(* CoDeSys 2.3 export: UDP_COMMUNICATION.EXP *)
(* Libraries: 05_Utilities\MPLCCommunication_Ethernet.lib 30.1.17 00:00:00, 11_System\SysLibSockets.lib 27.1.17 13:50:06, Internal\MPLCIntern_Communication_Ethernet.lib 30.1.17 00:00:00, standard.lib 27.1.17 13:50:06 *)

(* Global variable list: CodeSamples/UDP_Communication/UDP_Konstanten *)
VAR_GLOBAL CONSTANT
	UDP_CommAnzPD: INT := 64;  (*Datengröße in Byte*)
END_VAR
VAR_GLOBAL
END_VAR

(* POU CodeSamples/UDP_Communication/UDP_Communication_PRG, FBD *)
PROGRAM UDP_Communication_PRG
VAR
	bTest1: BOOL;
	bTest2: BOOL;
	bTest3: BOOL;
	fbUDP_Communication_MasterSlave: UDP_Communication_MasterSlave;
	bMaster: BOOL;
	nPort: UINT;
	sIP: STRING;
	tCycleTime: TIME;
	DataOUT: ARRAY[1..UDP_CommAnzPD] OF WORD;
	ttimeOut: TIME;
	DataIN: ARRAY[1..UDP_CommAnzPD] OF WORD;
END_VAR

(*Example inputs for MASTER---------------------------------------------------------------
UDP_Communication_MasterSlave(
	Enable:=TRUE , 
	SendMaster:=TRUE , 
	Port:= 44818, 
	IPAdr:= '10.1.254.129', 
	CycleTime:=t#100ms, 
	PE_Data:=fbUDP_Communication_MasterSlave.PE_Data , 
	TimeOut:=t#1000ms , 
	ChangeByteOrder:=FALSE , 
	Done=> , 
	Error=> , 
	ErrorID=> , 
	PDTimeOut=> , 
	PA_Data=> );

Example inputs for SLAVE---------------------------------------------------------------
UDP_Communication_MasterSlave(
	Enable:=TRUE , 
	SendMaster:=FALSE , 
	Port:= 44818, 
	IPAdr:= '10.1.254.128', 
	CycleTime:=t#100ms, 
	PE_Data:=fbUDP_Communication_MasterSlave.PE_Data , 
	TimeOut:=t#1000ms , 
	ChangeByteOrder:=FALSE , 
	Done=> , 
	Error=> , 
	ErrorID=> , 
	PDTimeOut=> , 
	PA_Data=> );
*)	
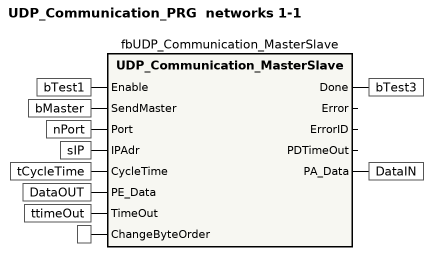
_FBD_ (* Function Block Diagram *)
NETWORK 1
	fbUDP_Communication_MasterSlave:UDP_Communication_MasterSlave(Enable: bTest1, SendMaster: bMaster, Port: nPort, IPAdr: sIP, CycleTime: tCycleTime, PE_Data: DataOUT, TimeOut: ttimeOut, ChangeByteOrder: , PA_Data => DataIN) => bTest3
_END_FBD_
END_PROGRAM

(* POU CodeSamples/UDP_Communication/UDP_Communication_MasterSlave, FBD *)
FUNCTION_BLOCK UDP_Communication_MasterSlave
VAR_INPUT
	Enable:BOOL;
	SendMaster : BOOL;  (* TRUE : Senden alle CycleTime, FALSE: Senden wenn ein Telegramm empfangen wurde *)
	Port:UINT;
	IPAdr:STRING(15);
	CycleTime :TIME;
	PE_Data:ARRAY[1..UDP_CommAnzPD] OF WORD;
	TimeOut:TIME;
	ChangeByteOrder : BOOL;
END_VAR
VAR_OUTPUT
	Done:BOOL;
	Error:BOOL;
	ErrorID:DWORD;
	PDTimeOut:BOOL;
	PA_Data:ARRAY[1..UDP_CommAnzPD] OF WORD;
END_VAR
VAR
	fbMC_ConnectV2_UDP: MC_ConnectV2_UDP;
	fbMC_ReceiveV2_UDP: MC_ReceiveV2_UDP;
	fbMC_SendV2_UDP: MC_SendV2_UDP;
	fbConvert_Array_1: WORDARRAY_TO_BYTEARRAY;
	fbConvert_Array: BYTEARRAY_TO_WORDARRAY_V2;
	R_TRIG_SendTrigger: R_TRIG;
	TON_TimeOut: TON;
	TON_CyclicSend: TON;

	refUDPConnection: MC_ConnectionV2_UDP;

	Send_Data_Array: ARRAY[0..1447] OF BYTE;
	Receive_Data_ArraY: ARRAY[0..1447] OF BYTE;


	bInitError: BOOL;
	nInitErrorID: DWORD;
	bSendError: BOOL;
	nSendErrorID: DWORD;
	bRecError: BOOL;
	nRecErrorID: DWORD;


	bCyclicSendTrigger: BOOL;
	bRecvDone: BOOL;

	nRxCounterOld: UINT;

END_VAR
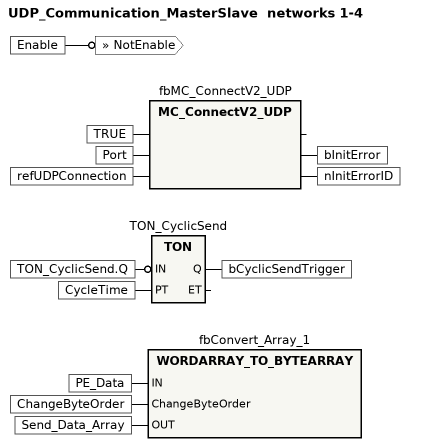
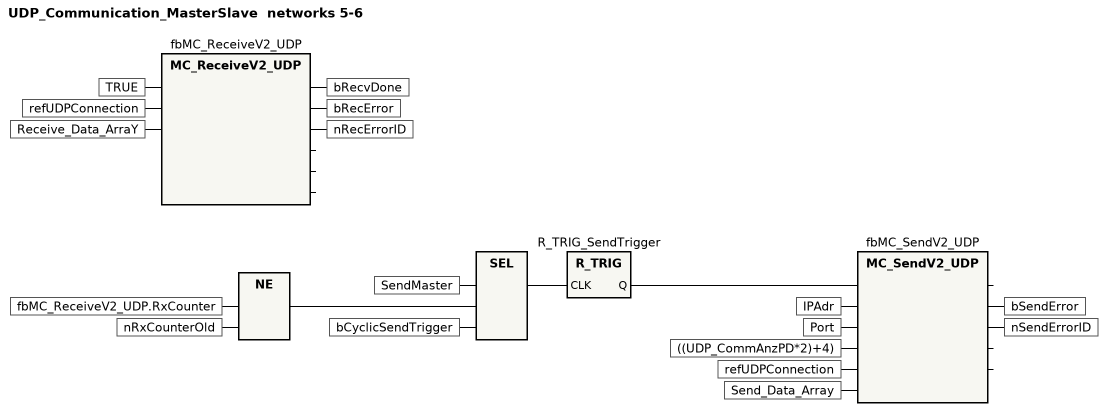
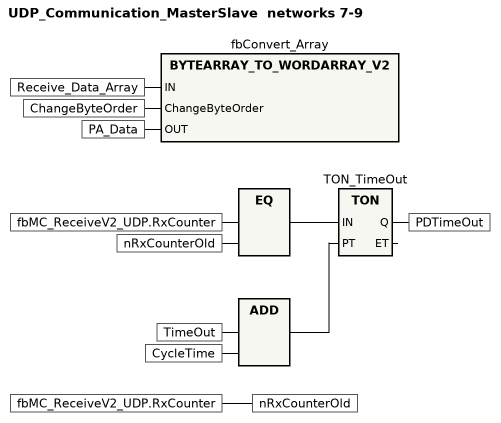
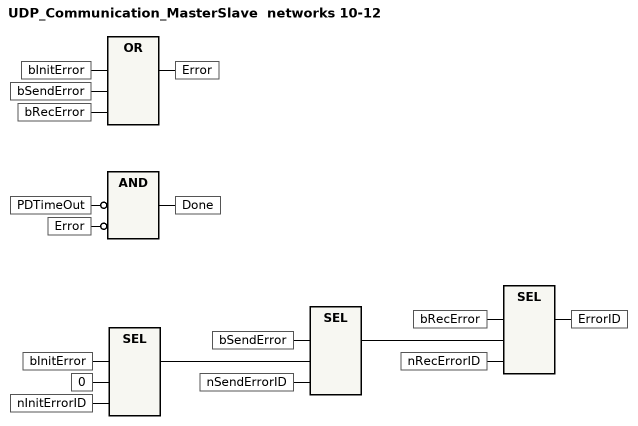
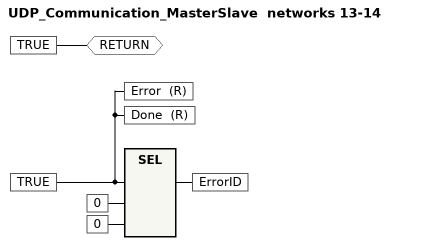
_FBD_ (* Function Block Diagram *)
NETWORK 1
	NOT Enable => >>NotEnable
NETWORK 2 (* Initialisierung der UDP-Kommunikation *)
	fbMC_ConnectV2_UDP:MC_ConnectV2_UDP(TRUE, Port, refUDPConnection, out 2 => bInitError, out 3 => nInitErrorID)
NETWORK 3 (* SendeTrigger für Senden wenn Master *)
	TON_CyclicSend:TON(IN: NOT TON_CyclicSend.Q, PT: CycleTime) => bCyclicSendTrigger
NETWORK 4 (* Umkopieren WORD-Array in BYTE-Array *)
	fbConvert_Array_1:WORDARRAY_TO_BYTEARRAY(IN: PE_Data, ChangeByteOrder: ChangeByteOrder, OUT: Send_Data_Array)
NETWORK 5 (* Daten empfangen über UDP *)
	fbMC_ReceiveV2_UDP:MC_ReceiveV2_UDP(TRUE, refUDPConnection, Receive_Data_ArraY, out 2 => bRecError, out 3 => nRecErrorID) => bRecvDone
NETWORK 6 (* Daten senden über UDP *)
	fbMC_SendV2_UDP:MC_SendV2_UDP(R_TRIG_SendTrigger:R_TRIG(CLK: SEL(SendMaster, NE(fbMC_ReceiveV2_UDP.RxCounter, nRxCounterOld), bCyclicSendTrigger)), IPAdr, Port, ((UDP_CommAnzPD*2)+4), refUDPConnection, Send_Data_Array, out 2 => bSendError, out 3 => nSendErrorID)
NETWORK 7 (* Konvertiere BYTE-Array in WORD-Array *)
	fbConvert_Array:BYTEARRAY_TO_WORDARRAY_V2(IN: Receive_Data_Array, ChangeByteOrder: ChangeByteOrder, OUT: PA_Data)
NETWORK 8
	TON_TimeOut:TON(IN: EQ(fbMC_ReceiveV2_UDP.RxCounter, nRxCounterOld), PT: ADD(TimeOut, CycleTime)) => PDTimeOut
NETWORK 9
	fbMC_ReceiveV2_UDP.RxCounter => nRxCounterOld
NETWORK 10 (* Errorbit setzen *)
	OR(bInitError, bSendError, bRecError) => Error
NETWORK 11
	AND(NOT PDTimeOut, NOT Error) => Done
NETWORK 12
	SEL(bRecError, SEL(bSendError, SEL(bInitError, 0, nInitErrorID), nSendErrorID), nRecErrorID) => ErrorID
NETWORK 13
	TRUE => <RETURN>
NETWORK 14 NotEnable: (* Comment *)
	SEL(<TRUE => R Error, R Done>, 0, 0) => ErrorID
_END_FBD_
END_FUNCTION_BLOCK

(* POU CodeSamples/UDP_Communication/Subroutines/WORDARRAY_TO_BYTEARRAY, ST *)
FUNCTION_BLOCK WORDARRAY_TO_BYTEARRAY
VAR
	Data_H	:BYTE;
	Data_L	:BYTE;
	a			:INT;
END_VAR
VAR_INPUT
	IN					:ARRAY [1..UDP_CommAnzPD] OF WORD;
	ChangeByteOrder	:BOOL;
END_VAR
VAR_IN_OUT
	OUT		:ARRAY [0..1447] OF BYTE;
END_VAR
FOR a:=0 TO (UDP_CommAnzPD-1) DO
	Data_L:= WORD_TO_BYTE(IN[a+1]);
	Data_H:=WORD_TO_BYTE(SHR(IN[a+1],8));

	IF ChangeByteOrder THEN	(*Tausche High-Byte und Low-Byte z.B.: für S7 Kommunikation*)
		OUT[a*2]:=Data_H;
		OUT[a*2+1]:=Data_L;
	ELSE
		OUT[a*2]:=Data_L;
		OUT[a*2+1]:=Data_H;
	END_IF
END_FOR
END_FUNCTION_BLOCK

(* POU CodeSamples/UDP_Communication/Subroutines/BYTEARRAY_TO_WORDARRAY_V2, ST *)
FUNCTION_BLOCK BYTEARRAY_TO_WORDARRAY_V2
VAR
	a		:INT;
	Data	:WORD;
END_VAR
VAR_INPUT
	IN		:ARRAY [0..1447] OF BYTE;
	ChangeByteOrder: BOOL;	(*  *)
END_VAR
VAR_IN_OUT
	OUT	:ARRAY [1..UDP_CommAnzPD] OF WORD;
END_VAR
FOR a:= 0 TO ((UDP_CommAnzPD*2)-1) BY 2 DO

	(*Data:= IN[a] + SHL(IN[a+1], 8); old until 2014-01-24, SHL 8 with a BYTE variable erases all data and creates zero*)
	Data:= IN[a] + SHL(BYTE_TO_WORD(IN[a+1]), 8);

	IF ChangeByteOrder THEN	(*Tausche High-Byte und Low-byte z.B.: für S7-Kommunikation*)
	Data:=ROL(Data,8);
	END_IF

	OUT[((a+1)/2)+1]:=Data;
END_FOR
END_FUNCTION_BLOCK
